PROGRAM Func_block_example
VAR
	myCounter : CTU;
	bCountUp: BOOL;
	bReset: BOOL;
	bCountDone: BOOL;
	myPulse : FB_Pulse;
	myPulse2 : FB_Pulse;
END_VAR

myCounter(
	CU:= bCountUp,
	RESET := bReset,
	PV:= 5, 
	Q=>bCountDone , 
	CV=> );
	
	
myPulse(bEnable:= , tTimeOn:= T#1S, tTimeOff:= T#500MS, bPulse=> );

myPulse2();

END_PROGRAM

(* stored: Version 1.1.0.1, ProductVersion 3.1.4024.9
   POU Func_block_example: Id {f2f70ce4-cadd-4305-b209-15899cc09469}, SpecialFunc None *)
